// TIA Portal project "Tram1_full" (V16)

(* hardware
DEVICE "S7-1200 station_1"  S7-1200 Station
   slot 0: "Rack_0"  S7-1200 Rack  Rack  V1.0
   slot 1: "PLC_1"  CPU 1214C DC/DC/DC  6ES7 214-1AG40-0XB0  V4.1
   slot 2: "DQ 16xRelay_1"  SM 1222 DQ16 x relay  6ES7 222-1HH32-0XB0  V2.0
DEVICE "HMI_1"  KTP400 Basic PN
   slot 0: "HMI_1"  KTP400 Basic PN  6AV2 123-2DB03-0AX0  15.0.0.0
   slot 1: "HMI_RT_1"  KTP400 Basic PN  6AV2 123-2DB03-0AX0  15.0.0.0
   slot 5: "HMI_1.IE_CP_1"  PROFINET Interface  15.0.0.0
      slot 1: "PROFINET Interface_1"  PROFINET Interface
         slot 1: "Port_1"  Port
*)

// ===== PLC "PLC_1"  CPU 1214C DC/DC/DC =====

VAR_GLOBAL   // PLC tag table "Default tag table"
   "RED" AT %Q9.7 : Bool;
   "GREEN" AT %Q9.6 : Bool;
   "START" AT %I0.0 : Bool;
   "STOP" AT %I0.1 : Bool;
   "Motor" AT %Q9.2 : Bool;
   "Tag_6" AT %M0.1 : Bool;
   "Tag_8" AT %M0.0 : Bool;
   "SQ1" AT %I0.2 : Bool;
   "SQ2" AT %I0.3 : Bool;
   "CLY1" AT %Q9.5 : Bool;
   "Tag_7" AT %M0.2 : Bool;
   "SQ3" AT %I0.4 : Bool;
   "Tag_1" AT %Q9.1 : Bool;
END_VAR

// folder: System blocks/Program resources

DATA_BLOCK "C1"   // DB2
{ S7_Optimized_Access := 'TRUE' }
AUTHOR : Simatic
FAMILY : IEC
NAME : CNTR
VERSION : 1.0
// stored: InstanceOfName IEC_COUNTER
"IEC_COUNTER"
BEGIN
END_DATA_BLOCK

DATA_BLOCK "T2"   // DB3
{ S7_Optimized_Access := 'TRUE' }
AUTHOR : Simatic
FAMILY : IEC
NAME : IEC_TMR
VERSION : 1.0
// stored: InstanceOfName IEC_TIMER
"IEC_TIMER"
BEGIN
END_DATA_BLOCK

// folder: (top level)

ORGANIZATION_BLOCK "Main_1"   // OB123, LAD, ProgramCycle
TITLE = "Main Program Sweep (Cycle)"
{ S7_Optimized_Access := 'TRUE' }
VERSION : 0.1
   VAR_INPUT
      Initial_Call : Bool;   // Initial call of this OB
      Remanence : Bool;   // =True, if remanent data are available
   END_VAR
   VAR_TEMP   // added for the SCL form of the ladder/FBD networks
      _w1 : Bool;
   END_VAR
BEGIN

REGION Network 1
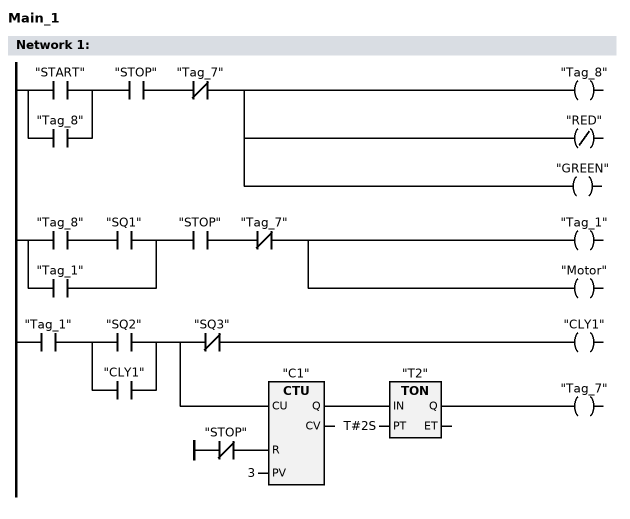
   "Tag_8" := ("START" OR "Tag_8") AND "STOP" AND NOT "Tag_7";
   "RED" := NOT "Tag_8";
   "GREEN" := "Tag_8";
   "Tag_1" := (("Tag_8" AND "SQ1") OR "Tag_1") AND "STOP" AND NOT "Tag_7";
   "Motor" := "Tag_1";
   #_w1 := "Tag_1" AND ("SQ2" OR "CLY1");
   "CLY1" := #_w1 AND NOT "SQ3";
   "C1".CTU(CU := #_w1, R := NOT "STOP", PV := 3);
   "T2".TON(IN := "C1".Q, PT := T#2S);
   "Tag_7" := "T2".Q;
END_REGION
END_ORGANIZATION_BLOCK

(* ===== HMI "HMI_RT_1" =====
system functions are stored by id; their names below are inferred from use
connection "HMI_Connection_1": ETHERNET, SMART_S7_1200_OMS

HMI tags "Default tag table"
   "Tag_ScreenNumber" : UInt, internal
   "Tag_9" : Bool = PLC Tag_9 AT %I0.0, 1 s

Template "Template_1" 480x272
   Button "Exit" at 388,227 size 63x44; TextOff 'Exit'; PictureOff "ExitRuntime_KTP400_Basic_PN_TR"; PictureOn "ExitRuntime_KTP400_Basic_PN_TR"
      on Release: StopRuntime(0)
   Button "Template_Button" at 268,227 size 63x44; TextOff 'Text'
   Button "Alarms" at 148,227 size 63x44; TextOff 'Alarms'; PictureOff "AlarmDisplay_KTP400_Basic_PN_TR"; PictureOn "AlarmDisplay_KTP400_Basic_PN_TR"
      on Release: function_ef3f5d25("Alarm window_Unacknowledged", -1)
   Button "Start screen" at 28,227 size 63x44; TextOff 'Start screen'; PictureOff "NavigateHome_KTP400_Basic_PN_TR"; PictureOn "NavigateHome_KTP400_Basic_PN_TR"
      on Release: ActivateScreen("Root screen", 0)
   SymbolicIOField "Symbolic_IO_Field_Screen" at 82,8 size 311x29; TextOff '0'; TextOn '1'; TextList "TextList_ScreenNames"
      ProcessValue <- "Tag_ScreenNumber"
      on Change: ActivateScreenByNumber("Tag_ScreenNumber", 0)
   DateTimeField "HmiScreenItemData" at 395,22 size 85x22
   DateTimeField "HmiScreenItemData_1" at 395,0 size 85x22
   GraphicView "Logo" at 0,0 size 80x45; Picture "Logo of HMI_1"

screen "Root screen" 480x272, template "Template_1"
   on GenerateScreen: SetTag("Tag_ScreenNumber", 1)
   TextField "HmiScreenItemData" at 48,122 size 384x22; Text 'Welcome to HMI_1 (KTP400 Basic+ PN)!'

screen "Screen_1" 480x272
   Circle "Circle_1" at 50,50 size 48x48
      Appearance <- "Tag_9"
   Button "Button_1" at 177,49 size 111x49; TextOff 'Text'
      on Press: SetBit("Tag_9")
      on Release: SetBit("Tag_9")
*)